// TIA Portal V16 export
// export: Created 2019-09-22T13:16:38.7801748Z, ExportSetting WithDefaults, DisplayName Totally Integrated Automation Portal, DisplayVersion V16, DisplayName TIA Portal Version Control Interface, DisplayVersion V16, DisplayName TIA Portal Openness, DisplayVersion V16, DisplayName STEP 7 Professional, DisplayVersion V16, DisplayName SIMATIC Energy Suite, DisplayVersion V16, DisplayName STEP 7 Safety, DisplayVersion V16, DisplayName WinCC Professional, DisplayVersion V16, DisplayName SIMATIC Visualization Architect, DisplayVersion V16
DATA_BLOCK "SeqData"   // DB15
{ S7_Optimized_Access := 'TRUE' }
VERSION : 0.1
// stored: AutoNumber true, DBAccessibleFromOPCUA true, IsOnlyStoredInLoadMemory false, IsRetainMemResEnabled false, IsWriteProtectedInAS false, MemoryReserve 100
   VAR
      plantOn : Bool := true;   // Plant switched on
      compressedAir : Bool;   // Druckluft OK / Compressed air OK
      powerVoltage : Bool;   // Power voltage OK
      doorClosed : Bool;   // Schutztür geschlossen / Safety door closed
      autoStart : Bool := true;   // Automatic start
      autoStarted : Bool;   // Automatic started
      autoStopped : Bool;   // Automatic stopped
      ackSeq : Bool;   // Acknowledge GRAPH FB
      errFltSeq : Bool;   // Error Graph FB / Fehler Graph FB
      seqStart : Bool;   // GRAPH sequence started
      newCase : Bool;   // Sensor new case
      posCaseBelt : Int;   // Case position on belt
      posLift1 : Int;   // Lift 1 position
      posLift2 : Int;   // Lift 2 position
      visCaseLift1 : Bool;   // Case lift1 visible
      visCaseLift2 : Bool;   // Case lift2 visible
      startLift1Up : Bool;   // Start lift1 up
      startLift1Down : Bool;   // Start lift1 down
      startLift2Up : Bool;   // Start lift2 up
      startLift2Down : Bool;   // Start lift2 down
      setStop1 : Bool;   // Set stopper1
      setStop2 : Bool;   // Set stopper2
      sensorStop1 : Bool;   // Sensor at stopper1
      sensorStop2 : Bool;   // Sensor at stopper2
      sensorStop3 : Bool;   // Sensor at stopper3
      errSensorStop1 : Bool;   // Error at sensor stopper 1 / Fehler bei Stopper 1
      errSensorStop2 : Bool;   // Error at sensor stopper 1 / Fehler bei Stopper 1
      errSensorStop3 : Bool;   // Error at sensor stopper 1 / Fehler bei Stopper 1
      errSensorNewCase : Bool;   // Error at sensor new case / Fehler bei Sensor "Neues Case"
      sensorLift1Top : Bool;   // Sensor lift1 up
      sensorLift1Bottom : Bool;   // Sensor lift1 down
      sensorLift2Top : Bool;   // Sensor lift2 up
      sensorLift2Bottom : Bool;   // Sensor lift2 down
      toLift1 : Bool;   // Case to lift1 or lift2
      outLift1Up : Bool;   // Output lift1 up
      outLift1Down : Bool;   // Output lift1 down
      outLift2Up : Bool;   // Output lift2 up
      outLift2Down : Bool;   // Output lift2 down
      manLift1Up : Bool;   // Manual start lift1 up
      manLift1Down : Bool;   // Manual start lift1 down
      manLift2Up : Bool;   // Manual start lift2 up
      manLift2Down : Bool;   // Manual start lift2 down
      simOperandSupVis : Bool;   // Simulation supervision operand
      simInterlockSupVis : Bool;   // Simulation supervision interlock
      simActReactSupVis : Bool;   // Simulation supervision action and reaction
      simPositionSupVis : Bool;   // Simulation supervision position
      simActive : Bool;   // Simulation aktiv / Simulation active
      releaseSimPlantOn : Bool;   // Release simulation plant on
      stateCase : Array[0..3] of Bool;   // State case position
      liftBlocked : Bool;   // Lift is blocked / Lift ist bereit für einen neuen Kasten
      resetCrit : Bool;   // Reset initial value acquisition
   END_VAR
BEGIN
END_DATA_BLOCK
